{attribute 'GeneratedUsingTerminal: KL3361-0001'}
{attribute addProperty BoxType "KL3361-0001"}
{attribute addProperty Id "Channel_1AT %Q*Channel_3C1A65000"}
{attribute addProperty CRC "3994895622"}
{attribute addProperty Size "0"}
TYPE KL_EE1D4506 :
STRUCT
	{attribute addProperty Name "Channel_1"}
	Channel_1 : Channel_3C1A6500;
END_STRUCT
END_TYPE

(* stored: Version 1.2.0.0, ProductVersion 3.1.4024.9
   DUT KL_EE1D4506: Id {85593a36-de5b-4169-b273-4045132ce8f0} *)
